# B&R Automation Studio project LibUserLog
Automation Studio 4.9.3.144 SP; Sample project for the UserLog library

## Configuration ARM

CPU X20CP0484, AutomationRuntime 6.7.5, Build 11.3.0

### Task classes (Cpu.sw)
```
Binaries: udbdef, TCLang, TCData, arconfig, TC, asfw, ashwac, ashwd, sysconf
Libraries: UserLog, ArEventLog, runtime, sys_lib, astime, ArEventLog, sys_lib, astime, runtime
```

### Hardware
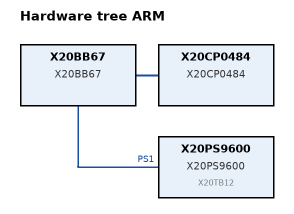
```
X20BB67 : X20BB67 v1.3.1.0
X20CP0484 : X20CP0484 v1.8.1.0  [SL -> X20BB67.SL1]
  Connector IF2:
    ActivateDevice = 1
    InaPort = 11160
  ConfigurationID = UserLogProject_ARM
  TimerDeviceType = SWIOTIMER
  Cyclic1Duration = 10000
  Cyclic1Tolerance = 10000
  Cyclic2Duration = 20000
  Cyclic2Tolerance = 20000
  Cyclic3Duration = 50000
  Cyclic3Tolerance = 50000
  Cyclic4Duration = 100000
  Cyclic4Tolerance = 100000
  Cyclic5Duration = 200000
  Cyclic5Tolerance = 200000
  Cyclic6Duration = 500000
  Cyclic6Tolerance = 500000
  Cyclic7Duration = 1000000
  Cyclic7Tolerance = 1000000
  Cyclic8Duration = 10000
  Cyclic8Tolerance = 30000000
  FileDevice1
  FileDeviceName1 = USER
  FileDevicePath1 = USER_PATH
  ActivateFtpServer = 1
  ActivateWebServer = 1
  ActivateSdm = 1
X20PS9600 : X20PS9600 v1.6.2.0  [PS -> X20BB67.PS1; SS1 -> X20TB12.SS]
X20TB12 : X20TB12 v1.0.0.0
```

## Configuration Config1

CPU X20CP1586, AutomationRuntime C4.90, Build 4.1.2, Vc 

### Task classes (Cpu.sw)
```
Cyclic#1:
  Develop <- (binary)
  EventLog <- (binary)
Binaries: FWRules, TCData, udbdef, asfw, User, iomap, sysconf, arconfig, ashwd, Role, ashwac, TCLang, TC
Libraries: ArEventLog, UserLog, sys_lib, asieccon, astime, MathTools, Library
```

### Hardware
```
X20CP1586 : X20CP1586 v1.10.0.0
  Connector IF1:
    ActivateIna = 0
  Connector IF2:
    ActivateDevice = 1
    InaPort = 11160
  ConfigurationID = UserLogPrj_Simulation
```

## Configuration Config2

CPU X20CP0484, AutomationRuntime C4.90, Build 4.1.2, Vc 

### Hardware
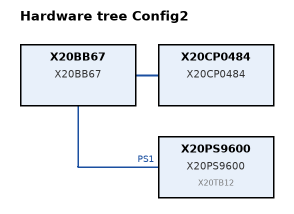
```
X20BB67 : X20BB67 v1.2.0.0
X20CP0484 : X20CP0484 v1.5.0.0  [SL -> X20BB67.SL1]
  Connector IF2:
    ActivateDevice = 1
    InaPort = 11160
  ConfigurationID = UserLogPrj_Simulation
  TimerDeviceType = SWIOTIMER
  Cyclic1Duration = 10000
  Cyclic1Tolerance = 10000
  Cyclic2Duration = 20000
  Cyclic2Tolerance = 20000
  Cyclic3Duration = 50000
  Cyclic3Tolerance = 50000
  Cyclic4Duration = 100000
  Cyclic4Tolerance = 100000
  Cyclic5Duration = 200000
  Cyclic5Tolerance = 200000
  Cyclic6Duration = 500000
  Cyclic6Tolerance = 500000
  Cyclic7Duration = 1000000
  Cyclic7Tolerance = 1000000
  Cyclic8Duration = 10000
  Cyclic8Tolerance = 30000000
X20PS9600 : X20PS9600 v1.6.0.0  [PS -> X20BB67.PS1; SS1 -> X20TB12.SS]
X20TB12 : X20TB12 v1.0.0.0
```

## Configuration Intel

CPU X20CP1586, AutomationRuntime T4.93, Build 6.3.0, Vc 

CPU X20CP1684, AutomationRuntime 6.7.6, Build 11.3.0

### Task classes (Cpu.sw)
```
Binaries: udbdef, TCLang, TCData, arconfig, TC, asfw, ashwac, ashwd, sysconf
Libraries: UserLog, IecString, ArEventLog, sys_lib, astime, runtime
```

### Hardware
```
X20CP1684 : X20CP1684 v1.9.0.0
  Connector IF1:
    ActivateIna = 0
  Connector IF2:
    ActivateDevice = 1
    InaPort = 11160
  ConfigurationID = UserLogProject_Intel
  FileDevice1
  FileDeviceName1 = USER
  FileDevicePath1 = USER_PATH
  ActivateFtpServer = 1
  ActivateWebServer = 1
  ActivateSdm = 1
```

## Configuration Simulation

CPU PC_any, AutomationRuntime C4.90, Build 4.1.2, Vc 

### Task classes (Cpu.sw)
```
Cyclic#1:
  EventLog <- LibArEventLog_ST.EventLog.prg
  Sample <- Sample.prg [disabled]
  Program <- Program.prg
Binaries: FWRules, TCData, udbdef, asfw, User, iomap, sysconf, arconfig, ashwd, Role, ashwac
Libraries: ArEventLog, runtime, AsBrStr, UserLog [disabled], asieccon, astime, Library, sys_lib
```

### Hardware
```
PC : PC_any v1.1.1.0 (OrderNumber=PC)
  ConfigurationID = UserLogPrj_Simulation
```

## Configuration UnitTest

CPU PC_any, AutomationRuntime 6.7.6, Build 11.3.0

### Task classes (Cpu.sw)
```
Cyclic#1:
  TestSuite <- Source.UnitTest.TestSuite.prg
Binaries: udbdef, TCLang, TCData, arconfig, TC, asfw, ashwac, ashwd, sysconf
Libraries: UserLog, IecString, ArEventLog, sys_lib, astime, runtime, UnitTest, UtMgr, UtWs, AsBrStr, AsARCfg, AsIecCon
```

### Hardware
```
PC : PC_any v1.1.2.0 (OrderNumber=PC)
  ConfigurationID = UserLogProject_UnitTest
  FileDevice1
  FileDeviceName1 = USER
  FileDevicePath1 = USER_PATH
  ActivateFtpServer = 1
  ActivateWebServer = 1
  ActivateSdm = 1
```

## Logical view

Binary libraries used (declarations not repeated): operator, runtime, astime, AsIecCon, ArEventLog, AsBrStr, UserLog, sys_lib

### Package Logical/Libraries - Global libraries

### Library Logical/Libraries/Library (IEC)

#### Library.fun - Exported functions and function blocks
```iecst
FUNCTION GetName : UINT
	VAR_INPUT
		TaskName : UDINT;
	END_VAR
END_FUNCTION
```

#### TaskName.st
```iecst
FUNCTION GetName

	GetName := ST_name(0, TaskName, 0);

END_FUNCTION
```

### Library Logical/Libraries/UnitTest (ANSIC, version 6.5.0) - Static library for UnitTest programs written in ANSI C /C++

#### UnitTest.h
```c
/*****************************************************************************
 * COPYRIGHT (C) BERNECKER + RAINER
 *****************************************************************************
 * Library:  UnitTest
 * File:     UnitTest.h
 * Author:   B+R
 *****************************************************************************
 * Description: Static library for UnitTest programs written in ANSI C /C++
 *
 * Add the path "\Logical\TS_UnitTest\Libraries\UnitTest\" to the
 * "Additional include directories" in the tab "Build" (PLC Properties)
 ******************************************************************************/

#ifndef	__UNITTEST_H__
#define	__UNITTEST_H__
#ifdef __cplusplus
extern "C"
{
#endif
#include <bur/plctypes.h>

#ifndef NULL
#define	NULL	0
#endif
#include "include/Test.h"

#include "include/TestCase.h"
#include "include/TestListener.h"
#include "include/TestResult.h"
#include "include/TestCaller.h"

#include "include/AssertImpl.h"
#include "include/HelperMacro.h"
#include "include/utRunner.h"

/* function is a test case */
#define _TEST 			static testStatusEnum

/* function is a setup */
#define _SETUP_TEST 	static testStatusEnum 	setupTest

/* function is a teardown */
#define _TEARDOWN_TEST 	static testStatusEnum 	teardownTest

/* function is a setup for whole test set */
#define _SETUP_SET		static testStatusEnum	setupSet

/* function is a teardown for whole test set */
#define _TEARDOWN_SET 	static testStatusEnum	teardownSet

/* function is a cyclic handler for test set */
#define _CYCLIC_SET		static void 			cyclicSetCaller

/* Skipped test case */
#define SKIP_TEST  		_TEST
/* Skip all test cases of set */
#define SKIP_TEST_SET

/* Dummies for smart edit autocompletion.
See AssertImpl.h for real macros used by the compiler  */
#ifdef _SMART_EDIT_DUMMY_

/* String comparison.
Returns true if the strings are equal. */
BOOL TEST_ASSERT_EQUAL_STRING(char *expected,char  *actual);
/* Wstring comparison.
Returns true if the WSTRINGS are equal. */
BOOL TEST_ASSERT_EQUAL_WSTRING(unsigned short *expected,unsigned short *actual);
 /* Compares two memory blocks.
Returns true if [size] bytes are equal. */
BOOL TEST_ASSERT_EQUAL_MEM(void *expected, void *actual,UDINT size);
/* Compares integer values. Usable for all integer types.
Avoid comparison of unsigned with signed types.
Returns true if they are equal.
Note: If different, values are reported as DINT values in the test report */
BOOL TEST_ASSERT_EQUAL_INT(expected, actual);

/* Compares REAL values with delta = (expected * TEST_FLOAT_PRECISION).
Returns true if (difference <= delta) */
BOOL TEST_ASSERT_EQUAL_REAL(REAL expected,REAL actual);
/* Compares REAL values with explicit delta.
Returns true if (difference <= delta) */
BOOL TEST_ASSERT_REAL_WITHIN(REAL delta, REAL expected, REAL actual);
/* Compares LREAL values with delta = (expected * TEST_DOUBLE_PRECISION).
Returns true if (difference <= delta) */
BOOL TEST_ASSERT_EQUAL_LREAL(LREAL expected,LREAL  actual);
/* Compares LREAL values with explicit delta.
Returns true if (difference <= delta) */
BOOL TEST_ASSERT_LREAL_WITHIN(LREAL delta, LREAL expected, LREAL actual);

/* Compares float values with delta = (expected * TEST_FLOAT_PRECISION).
Returns true if (difference <= delta) */
BOOL TEST_ASSERT_EQUAL_FLOAT(float expected, float actual);
/* Compares float values with explicit delta.
Returns true if (difference <= delta) */
BOOL TEST_ASSERT_FLOAT_WITHIN(float delta, float expected, float actual);
/* Compares double values with delta = (expected * TEST_DOUBLE_PRECISION).
Returns true if (difference <= delta) */
BOOL TEST_ASSERT_EQUAL_DOUBLE(double expected, double actual);
/* Compares double values with explicit delta.
Returns true if (difference <= delta) */
BOOL TEST_ASSERT_DOUBLE_WITHIN(double delta, double expected, double actual);

/* Returns true if pointer is null */
BOOL TEST_ASSERT_NULL(void *pointer);
/* Returns true if pointer is not null */
BOOL TEST_ASSERT_NOT_NULL(void *pointer);
/* Returns true, if condition evals to  true */
BOOL TEST_ASSERT_MESSAGE(condition, char *message);
/* Returns true, if condition evals to  true */
BOOL TEST_ASSERT(condition);

/* Returns always false */
BOOL TEST_FAIL(char *message);

/* Add a note to the test report */
void TEST_INFO(char *message);
/* Add a note with location information to the test report */
void TEST_INFO_POS(char *message);

#ifdef __cplusplus
/* Test if expression throws given exception.
Catches all other exceptions as failure.
Note: Available for C++ only */
void TEST_ASSERT_THROW(expression, type);

/* Fails if expression throws any exceptions.
Note: Available for C++ only*/
void TEST_ASSERT_NO_THROW(expression);
#endif

/* Adds a test function with description to the Testfixture.
See UNITTEST_FIXTURES() */
void new_TestFixture(char *name, _TEST function);

/* Adds a test function with description to the Testfixture.
This test will be skipped
See UNITTEST_FIXTURES() */
void skipTestFixture(char *name, _TEST function);

/* Defines the order of test cases.
Should look like this
UNITTEST_FIXTURES(fixtures)
{
	new_TestFixture("test_1",test_1),
	new_TestFixture("test_2",test_2),
	new_TestFixture("test_3",test_3)
}
*/
void UNITTEST_FIXTURES(fixtures)

/* Standard UnitTest caller without any setup / teardown methods*/
void UNITTEST_CALLER_TEST(caller, char *name, fixtures);

/* Standard UnitTest caller with macro setup / teardown for tests*/
void UNITTEST_CALLER_BASIC(caller, char *name, fixtures);

/* UnitTest caller with macro setup / teardown for tests and test set */
void UNITTEST_CALLER_SET(caller, char *name, fixtures);

/* UnitTest caller with macro setup / teardown for tests and test set and cylic*/
void UNITTEST_CALLER_COMPLETE(caller, char *name, fixtures);

/* UnitTest caller with explicit setup / teardown for suite */
void UNITTEST_CALLER_SET_EXPLICIT(caller,name,setupTest,teardownTest,fixtures, setupSuite, teardownSuite);

/* UnitTest caller with explicit setup / teardown for suite and cylic */
void UNITTEST_CALLER_COMPLETE_EXPLICIT(caller,name,setupTest,teardownTest,fixtures, setupSuite, teardownSuite, cyclicCaller);

/* Adds a test set with description to the fixture of test sets.
See UNITTEST_TESTSET_FIXTURES() */
void new_TestSet(testcaller);

/* Defines the order of test sets.
Should look like this
UNITTEST_TESTSET_FIXTURES(fixtures)
{
	new_TestSet(testSet_1),
	new_TestSet(testSet_2),
	new_TestSet(testSet_3)
}*/
void UNITTEST_TESTSET_FIXTURES(fixtures);

/* Defines the test set list handling structure*/
void UNTITTEST_TESTSET_HANDLER();

#endif /*_SMART_EDIT_DUMMY_*/

/*
 Use to declare Test set for use in list of test sets of test programm
 See usage in autogeneratedFile.c / FixtureOfTestSets.c
*/
#define UNITTEST_TESTSET_DECLARATION 	extern const TestCaller

/* Default factor for precision used to test if REAL / float values  are equal.
(0.00001f) */
#define TEST_FLOAT_PRECISION 	(0.00001f)
/* Default factor for precision used to test if LREAL / double values  are equal.
(1e - 12f) */
#define TEST_DOUBLE_PRECISION 	(1e-12f)

#if (__GNUC__ != 11) || (__GNUC_MINOR__ != 3) || (__GNUC_PATCHLEVEL__ != 0)
#error UnitTest is compiled with GCC version 11.3.0. To use UnitTest switch GCC version to 11.3.0 or import a different solution package
#endif

#define UNIT_TEST_LIBRARY_VERSION  			"6.5.0"

#ifdef __cplusplus
};
#endif

#include "include/asserts.hpp"

#endif/*__UNITTEST_H__*/
```

### Program Logical/Source/UnitTest/TestSuite (ANSIC)

#### main.c - Init, cyclic, exit code
```c
#include <UnitTest.h>
#include <UtMgr.h>
#include <string.h>

UtMgrTestSuite_typ test_suite;

void _INIT ProgramInit(void)
{
    memset(&test_suite, 0, sizeof(test_suite));
    strcpy(test_suite.Name, "UserLog_Tests");
    strcpy(test_suite.Description,
            "Test common and edges cases of all functions");
    test_suite.Type = utMgrTEST_TYPE_C;
    strcpy(test_suite.MetaInformation,
            "Test cases for UserLog library");
    utInit(&test_suite);
}

void _CYCLIC ProgramCyclic(void)
{
    utCyclic(&test_suite);
}

void _EXIT ProgramExit(void)
{
    utExit(&test_suite);
}
```

#### load.c - Set fixtures
```c
#include <UnitTest.h>

UNITTEST_TESTSET_DECLARATION basic_set;
UNITTEST_TESTSET_DECLARATION even_text_set;

UNITTEST_TESTSET_FIXTURES (utTestSets)
{
    new_TestSet(basic_set),
    new_TestSet(even_text_set)
};

UNTITTEST_TESTSET_HANDLER();
```

#### test_basic.c - Test UserLogBasic
```c
#include <UnitTest.h>
#include <UserLog.h>
#include <ArEventLog.h>
#include <stdint.h>
#include <stdbool.h>
#include <string.h>

_TEST test_basic_pass(void)
{
    TEST_ASSERT_EQUAL_INT(1, 1);

    TEST_DONE;
}

_TEST test_basic_fail(void)
{
    TEST_ASSERT_EQUAL_INT(1, 0);

    TEST_DONE;
}

_TEST test_basic_severity_success(void)
{
    /* Perform test */
    UserLogBasic(USERLOG_SEVERITY_SUCCESS, 1234, "Hello World!");

    /* Read details from logbook synchronously */
    /* Get logbook identifier */
    ArEventLogGetIdent_typ get_ident;
    memset(&get_ident, 0, sizeof(get_ident));
    strcpy(get_ident.Name, "$arlogusr");
    get_ident.Execute = true;
    ArEventLogGetIdent(&get_ident);
    if (get_ident.StatusID) {
        TEST_FAIL("ArEventLogGetIdent error");
        TEST_DONE;
    }

    /* Get latest record */
    ArEventLogGetLatestRecordID_typ get_latest_record;
    memset(&get_latest_record, 0, sizeof(get_latest_record));
    get_latest_record.Ident = get_ident.Ident;
    get_latest_record.Execute = true;
    ArEventLogGetLatestRecordID(&get_latest_record);
    if (get_latest_record.StatusID) {
        TEST_FAIL("ArEventLogGetLatestRecordID error");
        TEST_DONE;
    }

    /* Read record */
    ArEventLogRead_typ read_record;
    memset(&read_record, 0, sizeof(read_record));
    read_record.Ident = get_ident.Ident;
    read_record.RecordID = get_latest_record.RecordID;
    read_record.Execute = true;
    ArEventLogRead(&read_record);
    if (read_record.StatusID) {
        TEST_FAIL("ArEventLogRead error");
        TEST_DONE;
    }

    /* Read additional data */
    char message[256];
    memset(&message, 0, sizeof(message));
    ArEventLogReadAddData_typ read_data;
    memset(&read_data, 0, sizeof(read_data));
    read_data.Ident = get_ident.Ident;
    read_data.RecordID = get_latest_record.RecordID;
    read_data.AddData = (uint32_t)&message;
    read_data.BytesToRead = read_record.AddDataSize;
    read_data.Execute = true;
    ArEventLogReadAddData(&read_data);
    if (read_data.StatusID) {
        TEST_FAIL("ArEventLogReadAddData error");
        TEST_DONE;
    }

    TEST_ASSERT_EQUAL_STRING("Hello World!", message);

    TEST_DONE;
}

UNITTEST_FIXTURES(fixtures)
{
    new_TestFixture("UserLogBasic pass", test_basic_pass),
    new_TestFixture("UserLogBasic fail", test_basic_fail),
    new_TestFixture("UserLogBasic severity success",
                    test_basic_severity_success)
};

UNITTEST_CALLER_TEST (basic_set, "UserLogBasic test set", fixtures);
```

#### test_event_text.c - Test UserLogEventText
```c
#include <UnitTest.h>
#include <UserLog.h>
#include <ArEventLog.h>
#include <stdint.h>
#include <stdbool.h>
#include <string.h>

#define LOGBOOK_USER "$arlogusr"
#define SAMPLE_EVENT 1611615776
#define SAMPLE_BOOL 1
#define SAMPLE_FLOAT 4.56
#define SAMPLE_INT 7
#define SAMPLE_STRING "Hello World!"

#define GET_IDENT ArEventLogGetIdent_typ get_ident = {{0}}; \
strcpy(get_ident.Name, LOGBOOK_USER); \
get_ident.Execute = true; \
ArEventLogGetIdent(&get_ident); \
if (get_ident.StatusID) \
{ \
    TEST_FAIL("ArEventLogGetIdent error"); \
    TEST_DONE; \
}

_TEST test_event_text_sample(void)
{
    /* Perform test */
    int32_t record;
    UserLogFormatType FormatValues;
    FormatValues.b[0] = SAMPLE_BOOL;
    FormatValues.f[0] = SAMPLE_FLOAT;
    FormatValues.i[0] = SAMPLE_INT;
    strcpy((char*)&FormatValues.s[0], (char*)&SAMPLE_STRING);
    record = UserLogEventText(LOGBOOK_USER, SAMPLE_EVENT, 0, NULL, "%b %f %i %s", &FormatValues);

    /* Read details from logbook synchronously */
    GET_IDENT

    /* Get latest record */
    ArEventLogGetLatestRecordID_typ get_latest_record = {0};
    get_latest_record.Ident = get_ident.Ident;
    get_latest_record.Execute = true;
    ArEventLogGetLatestRecordID(&get_latest_record);
    if (get_latest_record.StatusID)
    {
        TEST_FAIL("ArEventLogGetLatestRecordID error");
        TEST_DONE;
    }

    /* Read record */
    ArEventLogRead_typ read_record = {0};
    read_record.Ident = get_ident.Ident;
    read_record.RecordID = get_latest_record.RecordID;
    read_record.Execute = true;
    ArEventLogRead(&read_record);
    if (read_record.StatusID)
    {
        TEST_FAIL("ArEventLogRead error");
        TEST_DONE;
    }

    /* Read description */
    char message[256] = {0};
    ArEventLogReadDescription_typ read_message = {0};
    read_message.Ident = get_ident.Ident;
    read_message.RecordID = get_latest_record.RecordID;
    read_message.TextBuffer = (UDINT)&message;
    read_message.TextBufferSize = sizeof(message);
    read_message.Execute = true;
    while(!read_message.Done && !read_message.Error){
        ArEventLogReadDescription(&read_message);
        if (read_message.StatusID || read_message.Error)
        {
            TEST_FAIL("ArEventLogReadDescription error");
            TEST_DONE;
        }
    }

    TEST_ASSERT(record > 0);
    TEST_ASSERT_EQUAL_INT(record, get_latest_record.RecordID);
    TEST_ASSERT_EQUAL_INT(SAMPLE_EVENT, read_record.EventID);

    /* Check description. Update this if the Sample tmx entry changes!! */
    char resultMessage[256] = {0};
    strcat((char*)&resultMessage, (char*)&"Sample UserLogEventText: ");
    strcat((char*)&resultMessage, (char*)&"TRUE ");
    strcat((char*)&resultMessage, (char*)&"4.560000 ");
    strcat((char*)&resultMessage, (char*)&"7 ");
    strcat((char*)&resultMessage, (char*)&SAMPLE_STRING);
    TEST_ASSERT_EQUAL_STRING(resultMessage, message);

    TEST_DONE;
}

UNITTEST_FIXTURES(fixtures)
{
    new_TestFixture("UserLogEventText success",
                    test_event_text_sample)
};

UNITTEST_CALLER_TEST (even_text_set, "UserLogEventText test set", fixtures);
```

### Program Logical/Source/ANSIC (ANSIC)

#### Main.c
```c
#ifdef _DEFAULT_INCLUDES
	#include <AsDefault.h>
#endif

#include <string.h>
#include <stdbool.h>

void _INIT ProgramInit(void)
{
	UserLogBasic(USERLOG_SEVERITY_SUCCESS, 1234, "Hello World!");

	FormatValues.b[0] = false;
	FormatValues.f[0] = 23.1;
	FormatValues.i[0] = -1070586087;
	strcpy(FormatValues.s[0], "Starting");
	UserLogAdvanced(USERLOG_SEVERITY_INFORMATION, 567, "Error=%b, Temperature=%f C, StatusID=%i, State=%s", &FormatValues);
    UserLogEventText("$arlogusr", USERLOG_EXAMPLE_TEXT_ID, 0, NULL, "%b %f %if %s", &FormatValues);

	UserLogCreate("Custom", 200000);
	UserLogCustom("Custom", USERLOG_SEVERITY_WARNING, 25, 789, 0, NULL, "This message is written to the Custom logbook", NULL);

	FormatValues.i[0] = UserLogSetSeverityLevel(USERLOG_SEVERITY_DEBUG);
	FormatValues.i[1] = USERLOG_SEVERITY_DEBUG;
	UserLogAdvanced(USERLOG_SEVERITY_DEBUG, 3, "Default severity level = %i, new severity level = %i", &FormatValues);

	UserLogSetSeverityLevel(USERLOG_SEVERITY_WARNING);
	UserLogBasic(USERLOG_SEVERITY_DEBUG, 1, "This is a debug message that will be suppressed");
	UserLogBasic(USERLOG_SEVERITY_WARNING, 2, "This is a warning message that will not be suppressed");

	Severity = UserLogGetSeverity(USERLOG_EXAMPLE_TEXT_ID);
	Facility = UserLogGetFacility(USERLOG_EXAMPLE_TEXT_ID);
	Code = UserLogGetCode(USERLOG_EXAMPLE_TEXT_ID);
}

void _CYCLIC ProgramCyclic(void)
{

}

void _EXIT ProgramExit(void)
{

}
```

### Program Logical/Source/IECST (IEC)

#### Main.st
```iecst
PROGRAM _INIT

	UserLogBasic(USERLOG_SEVERITY_SUCCESS, 1234, 'Hello World!');

	FormatValues.b[0] := FALSE;
	FormatValues.f[0] := 23.1;
	FormatValues.i[0] := -1070586087;
	FormatValues.s[0] := 'Starting';
    UserLogAdvanced(USERLOG_SEVERITY_INFORMATION, 567, 'Error=%b, Temperature=%f C, StatusID=%i, State=%s', FormatValues);
    UserLogEventText('$$arlogusr', USERLOG_EXAMPLE_TEXT_ID, 0, '', '%b %f %i %s', FormatValues);

	UserLogCreate('Custom', 200000);
	UserLogCustom('Custom', USERLOG_SEVERITY_WARNING, 25, 789, 0, '', 'This message is written to the Custom logbook', FormatValues);

	FormatValues.i[0] := UserLogSetSeverityLevel(USERLOG_SEVERITY_DEBUG);
	FormatValues.i[1] := USERLOG_SEVERITY_DEBUG;
	UserLogAdvanced(USERLOG_SEVERITY_DEBUG, 3, 'Default severity level = %i, new severity level = %i', FormatValues);

	UserLogSetSeverityLevel(USERLOG_SEVERITY_WARNING);
	UserLogBasic(USERLOG_SEVERITY_DEBUG, 1, 'This is a debug message that will be suppressed');
	UserLogBasic(USERLOG_SEVERITY_WARNING, 2, 'This is a warning message that will not be suppressed');

	Severity := UserLogGetSeverity(USERLOG_EXAMPLE_TEXT_ID);
	Facility := UserLogGetFacility(USERLOG_EXAMPLE_TEXT_ID);
	Code := UserLogGetCode(USERLOG_EXAMPLE_TEXT_ID);

END_PROGRAM

PROGRAM _CYCLIC

END_PROGRAM

PROGRAM _EXIT

END_PROGRAM
```

### Program Logical/Source/Sample (IEC)

#### Variables.var
```iecst
VAR
	LogCondition : BOOL;
	LogValues : UserLogFormatType;
END_VAR
```

#### Main.st
```iecst
PROGRAM _INIT

END_PROGRAM

PROGRAM _CYCLIC

	IF LogCondition THEN
		LogCondition := FALSE;
		UserLogAdvanced(USERLOG_SEVERITY_INFORMATION,
						123,
						'Error=%b, Temperature=%f C, StatusID=%i, State=%s',
						LogValues);
	END_IF

END_PROGRAM

PROGRAM _EXIT

END_PROGRAM
```

- UserLogText.csv - Text table (not shown)

- SetUserLogText.py - Convert csv to tmx (not shown)

### Global.typ - not listed in the package file held
```iecst
TYPE
	LogEntryType : 	STRUCT
		Severity : USINT;
		Code : UINT;
		sMessage : STRING[80];
	END_STRUCT;
	BufferEntryType : 	STRUCT
		LogEntry : LogEntryType;
		sTaskName : STRING[10];
	END_STRUCT;
END_TYPE
```

### Global.var - not listed in the package file held
```iecst
VAR
	WriteLogIndex : USINT;
	ReadLogIndex : USINT;
END_VAR
VAR CONSTANT
	MAX_LOG_INDEX : USINT := 9;
END_VAR
VAR
	LogBuffer : ARRAY[0..MAX_LOG_INDEX] OF BufferEntryType;
	LogBufferFull : BOOL;
END_VAR
```

### Program Logical/ANSIC

#### Variables.var
```iecst
VAR
	Logbook : STRING[10];
	Severity : UserLogSeverityEnum;
	Facility : UINT;
	Code : UINT;
	Origin : ArEventLogRecordIDType;
	Object : STRING[36];
	pObject : UDINT;
	Message : STRING[80];
	pMessage : UDINT;
	Arguments : UserLogFormatType;
	pArguments : UDINT;
	Test : BOOL;
	ReturnValue : ArEventLogRecordIDType;
	Level : UserLogSeverityEnum;
	TestLoop : BOOL;
	LoopMax : USINT;
	Index : USINT;
	EventID : DINT;
	GetSeverity : USINT;
	GetFacility : UINT;
	GetCode : UINT;
END_VAR
```

#### Main.c
```c
#include <bur/plctypes.h>
#include <string.h>
#include <stdint.h>
#include <stdbool.h>

#ifdef _DEFAULT_INCLUDES
	#include <AsDefault.h>
#endif

#define MAX(x,y) (((x) > (y)) ? (x) : (y))
#define MIN(x,y) (((x) < (y)) ? (x) : (y))

void _INIT ProgramInit(void)
{
	strcpy(Logbook, "$arlogusr");
	Severity = USERLOG_SEVERITY_DEBUG;
	Facility = 2;
	Code = 1234;
	pObject = (uint32_t)Object;
	strcpy(Message, "Hello World!");
	pMessage = (uint32_t)Message;
	pArguments = (uint32_t)&Arguments;
	Level = USERLOG_SEVERITY_SUCCESS;

	UserLogCreate("Test", 200000);

	UserLogBasic(USERLOG_SEVERITY_SUCCESS, 1234, "Hello World!");

	Arguments.i[0] = Code;
	UserLogAdvanced(USERLOG_SEVERITY_INFORMATION, Code, "My code is %i", &Arguments);

	LoopMax = 5;

	UserLogEventText("$arlogusr", USERLOG_EXAMPLE_TEXT_ID, 0, NULL, "This is a description of the log record", NULL);
}

void _CYCLIC ProgramCyclic(void)
{
	if(Test) {
		Test = false;
		ReturnValue = UserLogCustom(Logbook, Severity, Facility, Code, Origin, (char*)pObject, (char*)pMessage, (UserLogFormatType*)pArguments);
	}
	UserLogSetSeverityLevel(Level);

	if (TestLoop)
	{
		TestLoop = false;
		for (Index = 0; Index < LoopMax; Index++)
		{
			Arguments.i[0] = Index + 1;
			UserLogCustom(Logbook, Severity, Facility, Code, Origin, (char*)pObject, (char*)pMessage, (UserLogFormatType*)pArguments);
		}
	}

	EventID = ArEventLogMakeEventID(MIN(arEVENTLOG_SEVERITY_ERROR, MAX(arEVENTLOG_SEVERITY_SUCCESS, Severity)), Facility, Code);
	GetSeverity = UserLogGetSeverity(EventID);
	GetFacility = UserLogGetFacility(EventID);
	GetCode = UserLogGetCode(EventID);
}

void _EXIT ProgramExit(void)
{

}
```

### Program Logical/IECST

#### Variables.var
```iecst
VAR
	FormatValues : UserLogFormatType;
	Severity : USINT;
	Facility : UINT;
	Code : UINT;
END_VAR
```

#### Main.st
```iecst
PROGRAM _INIT

	UserLogBasic(USERLOG_SEVERITY_SUCCESS, 1234, 'Hello World!');

	FormatValues.b[0] := FALSE;
	FormatValues.f[0] := 23.1;
	FormatValues.i[0] := -1070586087;
	FormatValues.s[0] := 'Starting';
	UserLogAdvanced(USERLOG_SEVERITY_INFORMATION, 567, 'Error=%b, Temperature=%f C, StatusID=%i, State=%s', FormatValues);

	UserLogCreate('Custom', 200000);
	UserLogCustom('Custom', USERLOG_SEVERITY_WARNING, 25, 789, 0, '', 'This message is written to the Custom logbook', FormatValues);

	UserLogEventText('$$arlogusr', USERLOG_EXAMPLE_TEXT_ID, 0, '', 'This is a description of the log record', FormatValues);

	FormatValues.i[0] := UserLogSetSeverityLevel(USERLOG_SEVERITY_DEBUG);
	FormatValues.i[1] := USERLOG_SEVERITY_DEBUG;
	UserLogAdvanced(USERLOG_SEVERITY_DEBUG, 3, 'Default severity level = %i, new severity level = %i', FormatValues);

	UserLogSetSeverityLevel(USERLOG_SEVERITY_WARNING);
	UserLogBasic(USERLOG_SEVERITY_DEBUG, 1, 'This is a debug message that will be suppressed');
	UserLogBasic(USERLOG_SEVERITY_WARNING, 2, 'This is a warning message that will not be suppressed');

	Severity := UserLogGetSeverity(USERLOG_EXAMPLE_TEXT_ID);
	Facility := UserLogGetFacility(USERLOG_EXAMPLE_TEXT_ID);
	Code := UserLogGetCode(USERLOG_EXAMPLE_TEXT_ID);

END_PROGRAM

PROGRAM _CYCLIC

END_PROGRAM

PROGRAM _EXIT

END_PROGRAM
```

### Program Logical/Program

#### Variables.var
```iecst
VAR
	State : USINT;
	ErrorState : USINT;
	CmdLog : BOOL;
	EventID : DINT;
	Message : STRING[80];
	DataBuffer : ARRAY[0..81] OF USINT;
	SizeOfDataBuffer : UDINT;
	InitBufferReturn : BOOL;
	AddStringDataReturn : BOOL;
	fbGetIdent : ArEventLogGetIdent;
	fbWrite : ArEventLogWrite;
	StatusTaskName : UINT;
	sTaskName : STRING[31];
	UserLogIdent : ArEventLogIdentType;
END_VAR
```

#### Main.st
```iecst
(*******************************************************************************
 * Copyright: B&R Industrial Automation
 * Author:    Tyler Matijevich
 * Created:   October 28, 2020/16:30
********************************************************************************
 * Description: Test logging buffer code
********************************************************************************)

PROGRAM _INIT

	SizeOfDataBuffer := SIZEOF(DataBuffer);
	Message := 'Hello world! My name is Tyler.';
	StatusTaskName := GetName(ADR(sTaskName));

END_PROGRAM

PROGRAM _CYCLIC

	CASE State OF
		// INIT
		0:
			// Prepare the get ident FB
			fbGetIdent.Name := '$$arlogusr';
			fbGetIdent.Execute := TRUE;

			// Go to the next state
			State := 10;

		10:
			// Wait for compeletion
			IF fbGetIdent.Done THEN
				// Reset the FB
				fbGetIdent.Execute := FALSE;

				UserLogIdent := fbGetIdent.Ident;

				// Go to the next state
				State := 20;

			ELSIF fbGetIdent.Error THEN
				ErrorState := State;
				State := 255;

			END_IF

		1:
			IF CmdLog THEN
				CmdLog := FALSE;
				ErrorState := 0;

				// Create event ID
				EventID := ArEventLogMakeEventID(0, 1, 1001);

				// Initialize the data buffer
				InitBufferReturn := ArEventLogAddDataInit(ADR(DataBuffer), SizeOfDataBuffer, arEVENTLOG_ADDFORMAT_CODED);

				// Add string data to the buffer
				AddStringDataReturn := ArEventLogAddDataString(ADR(DataBuffer), SizeOfDataBuffer, ADR(Message));

				// Initialize the logbook ident
				fbGetIdent.Name := '$$arlogusr';
				fbGetIdent.Execute := TRUE;

				State := 10;

			END_IF

		11:
			IF fbGetIdent.Done THEN
				// Write to the logbook
				fbWrite.Ident := fbGetIdent.Ident;
				fbWrite.EventID := EventID;
				fbWrite.OriginRecordID := 0;
				fbWrite.AddDataSize := brsstrlen(ADR(Message));
				fbWrite.AddDataFormat := arEVENTLOG_ADDFORMAT_TEXT;
				fbWrite.AddData := ADR(Message);
				fbWrite.ObjectID := 'Sample';
				fbWrite.Execute := TRUE;

				State := 20;

			ELSIF fbGetIdent.Error THEN
				ErrorState := State;
				State := 255;

			END_IF

		21:
			IF fbWrite.Done THEN

				State := 0;

			ELSIF fbWrite.Error THEN
				ErrorState := State;
				State := 255;

			END_IF

		255:

	END_CASE

	// Call function blocks
	fbGetIdent();
	fbWrite();

END_PROGRAM

PROGRAM _EXIT

END_PROGRAM
```

### Program Logical/Sample

#### Variables.var
```iecst
VAR
	CmdWrite : BOOL;
	LogInfo : UserLogInfoType;
	InitReturn : DINT;
	InitReturn2 : DINT;
END_VAR
(*Burst example*)
VAR
	Run : BOOL;
	FormatArgs : FormatStringArgumentsType;
	MySeverity : UserLogSeverityEnum;
	MyCode : UINT;
	Index : USINT;
	NumOfMessages : USINT := 24;
	MyVerbosityLevel : UserLogSeverityEnum := USERLOG_SEVERITY_DEBUG;
END_VAR
```

#### Main.st
```iecst
(*******************************************************************************
 * File:      Sample\Main.st
 * Author:    Tyler Matijevich
 * Created:   October 20, 2020/20:34
********************************************************************************
 * Description: Demonstrate the functions and function blocks of the UserLog
 library
********************************************************************************)

PROGRAM _INIT

	// Initalize inputs to the LogMessage function
	MySeverity	:= USERLOG_SEVERITY_SUCCESS;
	MyCode 		:= 1001;

	InitReturn 	:= CreateCustomLogbook('MyLog', 200_000);
	InitReturn2	:= CreateCustomLogbook('MyLog2', 200_000);

END_PROGRAM

PROGRAM _CYCLIC

	// Write a single event to the User and custom logbook
	IF CmdWrite THEN
		CmdWrite := FALSE;
		LogMessage(MySeverity, MyCode, 'This message will be written to the User logbook');
		CustomMessage(MySeverity, MyCode, 'This message will be written to the MyLog logbook', 'MyLog', 1);
	END_IF

	// Write a burst of events to the user logbook. If it exceeds the max count, the events will be lost
	IF Run THEN
		Run := FALSE;
		// If loopMax is greater than USERLOG_MAX_MESSAGES then (loopMax - USERLOG_MAX_MESSAGES) number of entries will be lost
		// This can be observed in the log info structure
		// Increase USERLOG_MAX_MESSAGES if entries are found to be lost
		FOR Index := 1 TO NumOfMessages DO
			// Setup
			SetVerbosityLevel(MyVerbosityLevel);
			MySeverity := (Index - 1) MOD 6;
			MyCode := 1000 + Index;
			// Format
			FormatArgs.i[0] := Index;
			FormatArgs.i[1] := NumOfMessages;
			CASE MySeverity OF
				USERLOG_SEVERITY_CRITICAL: 		FormatArgs.s[0] := 'Critical';
				USERLOG_SEVERITY_ERROR: 		FormatArgs.s[0] := 'Error';
				USERLOG_SEVERITY_WARNING: 		FormatArgs.s[0] := 'Warning';
				USERLOG_SEVERITY_INFORMATION: 	FormatArgs.s[0] := 'Infomration';
				USERLOG_SEVERITY_SUCCESS: 		FormatArgs.s[0] := 'Success';
				USERLOG_SEVERITY_DEBUG: 		FormatArgs.s[0] := 'Debug';
			END_CASE
			// Log
			LogFormatMessage(MySeverity, MyCode, 'Event: %i of %i Severity: %s', FormatArgs);
		END_FOR
	END_IF

	GetUserLogInfo(LogInfo);

END_PROGRAM

PROGRAM _EXIT

END_PROGRAM
```

### Program Logical/String

#### Variables.var
```iecst
VAR
	str1 : STRING[10];
	str2 : STRING[12];
	mem1 : ARRAY[0..10] OF USINT;
	mem2 : ARRAY[0..12] OF USINT;
	formatArgs : FormatStringArgumentsType;
END_VAR
```

#### Main.c
```c
#include <bur/plctypes.h>
#include <string.h>

#ifdef _DEFAULT_INCLUDES
	#include <AsDefault.h>
#endif

void _INIT ProgramInit(void)
{
	strcpy(str2, "abcdefghijkl");
	memset(str1, 1, sizeof(str1));
	strncpy(str1, str2, sizeof(str1) - 1);
	memset(str1 + sizeof(str1) - 1, 0, 1);
	memcpy(mem1, str1, sizeof(mem1));
	memcpy(mem2, str2, sizeof(mem2));
}

void _CYCLIC ProgramCyclic(void)
{

}

void _EXIT ProgramExit(void)
{

}
```

### Program Logical/Test

#### Variables.var
```iecst
VAR
	Test : BOOL;
	Entries : UINT;
	Scans : UINT;
	IndexEntries : UINT;
	IndexScans : USINT;
	Args : FormatStringArgumentsType;
END_VAR
```

#### Main.st
```iecst
PROGRAM _INIT
	(* Insert code here *)
	LogMessage(severity := USERLOG_SEVERITY_SUCCESS, code := 1234, message := 'Hello World!');
END_PROGRAM

PROGRAM _CYCLIC
	(* Insert code here *)
	IF Test THEN
		FOR IndexEntries := 1 TO Entries DO
			Args.i[0] := IndexScans + 1;
			Args.i[1] := IndexEntries;
			LogFormatMessage(1, 1, 'Scan %i entry %i', Args);
		END_FOR

		IndexScans := IndexScans + 1;
		IF IndexScans >= Scans THEN
			Test := FALSE;
		END_IF
	ELSE
		IndexScans := 0;
	END_IF
END_PROGRAM

PROGRAM _EXIT
	(* Insert code here *)

END_PROGRAM
```

### Program Logical/Write

#### Variables.var
```iecst
VAR
	CmdWrite : BOOL;
	WriteCounter : INT;
	Message : STRING[80];
	Severity : USINT;
	Code : UINT;
	StatusTaskName : UINT;
	NextWriteIndex : USINT;
	sConstructMessage : STRING[80];
	MessageArguments : FormatStringArgumentsType;
	Facility : UINT;
END_VAR
```

#### Main.st
```iecst
(*******************************************************************************
 * Copyright: B&R Industrial Automation
 * Author:    Tyler Matijevich
 * Created:   October 29, 2020/15:57
********************************************************************************
 * Description: A short description
********************************************************************************)

PROGRAM _INIT

	Message := 'Test';
	Severity := 1;
	Code := 1001;

END_PROGRAM

PROGRAM _CYCLIC

	IF CmdWrite THEN
		CmdWrite := FALSE;

		IF LogBufferFull = FALSE THEN

			sConstructMessage := 'This is the log number %i';
			MessageArguments.i[0] := WriteCounter;
			IecFormatString(ADR(Message), 80, ADR(sConstructMessage), ADR(MessageArguments));
			WriteCounter := WriteCounter + 1;

			LogBuffer[WriteLogIndex].LogEntry.Severity 	:= Severity;
			LogBuffer[WriteLogIndex].LogEntry.Code		:= Code;
			LogBuffer[WriteLogIndex].LogEntry.sMessage 	:= Message;

			StatusTaskName := ST_name(0, ADR(LogBuffer[WriteLogIndex].sTaskName), 0);

			// Update write index
			WriteLogIndex := Math_WrapUSINT(WriteLogIndex + 1, 0, MAX_LOG_INDEX);
			IF WriteLogIndex = ReadLogIndex THEN
				LogBufferFull := TRUE;
			END_IF

		END_IF

	END_IF

END_PROGRAM

PROGRAM _EXIT

END_PROGRAM
```

Listed in the project but not available here: Logical/Libraries/Library/Types.typ, Logical/Libraries/Library/Constants.var, Logical/Libraries/UnitTest/include, Logical/Libraries/UnitTest/src
